PROGRAM CallHardware

//conveyors
callConveyors();

//robots
robot1();
robot2();
robot3();
robot4();
//robot5();
//robot6();

//A23
wrapperA23();

//A22
skidA22Left();
skidA22Right();
magazineA22Left();
magazineA22Right();

insertionA22Left(
	enable:= TRUE, 
	slider:= verticalDriveA22Left, 
	screw:= horizontalDriveA22Left, 
	contact=> , 
	active=> , 
	error=> , 
	home=> , 
	homingComplete=> , 
	sliderPos=> );
	
insertionA22Right(
	enable:= TRUE, 
	slider:= verticalDriveA22Right, 
	screw:= horizontalDriveA22Right, 
	contact=> , 
	active=> , 
	error=> , 
	home=> , 
	homingComplete=> , 
	sliderPos=> );
	
pistonA22Bottom();
wrapperA22();

//A21
skidA21Left();
skidA21Right();

magazineA21Left();
magazineA21Right();

stagingTableLeft();
stagingTableRight();

strapperA21();

insertionA21Left(
	enable:= TRUE, 
	slider:= verticalDriveA21Left, 
	screw:= horizontalDriveA21Left, 
	contact=> , 
	active=> , 
	error=> , 
	home=> , 
	homingComplete=> , 
	sliderPos=> );
	
insertionA21Right(
	enable:= TRUE, 
	slider:= verticalDriveA21Right, 
	screw:= horizontalDriveA21Right, 
	contact=> , 
	active=> , 
	error=> , 
	home=> , 
	homingComplete=> , 
	sliderPos=> );
	
pistonA21Bottom();

METHOD PRIVATE callConveyors : BOOL
VAR
	i : DINT;
END_VAR
//rewrite this method, call every conveyor individually
//calling via loop will not call derived implementations
(*
FOR i:=1 TO numConveyors BY 1 DO
	conveyorsArr[i]^(
		bEnable:= , 
		enable=> , 
		direction=> , 
		pulse=> , 
		reset=> , 
		error=> , 
		sensorEntry=> , 
		sensorExit=> , 
		requestLifter=> , 
		lifterEnable=> , 
		lifterDirection=> , 
		lifterPulse=> , 
		lifterReset=> , 
		lifterError=> , 
		extended=> , 
		retracted=> , 
		position=> , 
		velocity=> );
END_FOR
*)
END_METHOD

METHOD PRIVATE pushConveyorsToArray : BOOL
END_METHOD

END_PROGRAM

(* stored: Version 1.1.0.1, ProductVersion 3.1.4024.11
   POU CallHardware: Id {37cad5aa-fa76-4d83-b429-cad99db8cb21}, SpecialFunc None
   Method callConveyors: Id {365141b1-cb20-44d4-87c7-77ba15ac296c}
   Method pushConveyorsToArray: Id {cb74d2be-b24d-425a-bc95-cdcd1fdaeaaf} *)
